INTERFACE ITF_HMIManager EXTENDS ITF_BaseGroupElement

END_INTERFACE

(* stored: Version 1.1.0.1
   Itf ITF_HMIManager: Id {a317d999-660b-08b0-285a-99f61544469f} *)
